Universal Robots PolyScope program: a_to_d.urp

Program a_to_d (installation=string_planes directory=/programs/new folder_3 createdIn=5.17.3 lastSavedIn=5.17.3 robotSerialNumber=20245501435)
Calibrated DH parameters: a=[0.000154, -0.137004, -0.385524, -0.00002, 0.000092, 0]; d=[0.162441, 211.794786, -230.585024, 18.923638, 0.099786, 0.09951]; alpha=[1.569493, -0.001902, 0.003874, 1.570111, -1.570167, 0]; deltaTheta=[0, -1.242934, 1.056292, 0.186646, 0.000002, 0.000001]
InitVariablesNode
Robot Program (runOnlyOnce=false)
  MoveJ speed 60 deg/s, acceleration 80 deg/s^2 (useActiveTCP=true) feature=Base
    Waypoint Waypoint_9 (Relative): relativeFromPosition TCP in base x=327.369 y=541.717 z=231.872 mm, rx=1.6817 ry=2.3248 rz=-1.1114 rad; joints [-139.639, -50.321, 85.997, -84.695, -102.359, -153.08] deg; TCP offset x=28.21 y=-96.107 z=-99.69 mm, rx=0 ry=0 rz=0 rad; TCP in base x=337.287 y=452.573 z=146.265 mm, rx=-1.6084 ry=-2.1977 rz=1.0429 rad; joints [-146.228, -47.168, 100.748, -99.802, -91.44, -163.024] deg
